// TwinCAT 3 PLC project _25_Memento
// ProgramVersion: 3.1.4023.0
// libraries:
//   Tc2_Standard, * (Beckhoff Automation GmbH)
//   Tc2_System, * (Beckhoff Automation GmbH)
//   Tc3_Module, * (Beckhoff Automation GmbH)
// project tree:
//   / MAIN.TcPOU, PlcTask.TcTTO
//   Memento Pattern/FBs/ RecipeEditor.TcPOU, Snapshot.TcPOU
//   Memento Pattern/ P_Memento.TcPOU
// (motion and I/O tree: see PLC project 13_decorator)
// real-time tasks:
//   TASK PlcTask: cycle T#10ms, priority 20, ADS port 350
// variable links:

CONFIGURATION _25_Memento
    RESOURCE PLC ON TwinCAT3
        TASK PlcTask(INTERVAL := T#10ms, PRIORITY := 20);
        PROGRAM P_Memento WITH PlcTask : P_Memento;
    END_RESOURCE
END_CONFIGURATION

// ---- Memento Pattern/P_Memento.TcPOU
PROGRAM P_Memento
VAR
	// Recipe editor and backup object
	pBackup : POINTER TO Snapshot;
	editor : RecipeEditor;
	
	// Recipe settings
	sTitle: STRING := 'Recipe 1';
	sRecipeSteps : ARRAY[1..5] OF STRING := ['Move Home', 'Move To Station A', 'Heater On', 'Apply Heat', 'Heater Off'];
	
	// Demo program control values
	bSetValues	: BOOL;
	bMakeBackup : BOOL;
	bRestore	: BOOL;
END_VAR

// Set the recipe values
IF bSetValues THEN
	bSetValues := FALSE;
	editor.setRecipe(sRecipeSteps);
	editor.setTitle(sTitle);
END_IF

// Make a backup at any time
IF bMakeBackup THEN
	bMakeBackup := FALSE;
	pBackup := editor.createSnapshot();
END_IF

// Restore to the backup state
IF bRestore AND (pBackup <> 0)THEN
	bRestore := FALSE;
	pBackup^.restore();
END_IF

END_PROGRAM

// ---- Memento Pattern/FBs/Snapshot.TcPOU
{attribute 'enable_dynamic_creation'}
FUNCTION_BLOCK Snapshot
VAR
	pEditor : POINTER TO RecipeEditor;
	sTitle : STRING;
	sRecipeSteps : ARRAY[1..5] OF STRING;
END_VAR

METHOD FB_exit : BOOL
VAR_INPUT
	bInCopyCode : BOOL; // if TRUE, the exit method is called for exiting an instance that is copied afterwards (online change).
END_VAR
// Clear the pointer on exit
IF pEditor <> 16#0000 THEN
	pEditor := 16#0000;
END_IF
END_METHOD

METHOD FB_init : BOOL
VAR_INPUT
	bInitRetains : BOOL; // if TRUE, the retain variables are initialized (warm start / cold start)
	bInCopyCode : BOOL;  // if TRUE, the instance afterwards gets moved into the copy code (online change)
	pEditor : POINTER TO RecipeEditor;
	sTitle : STRING;
	sRecipeSteps : ARRAY[1..5] OF STRING;
END_VAR
THIS^.pEditor := pEditor;
THIS^.sTitle := sTitle;
THIS^.sRecipeSteps := sRecipeSteps;
END_METHOD

METHOD restore
VAR_INPUT
END_VAR
pEditor^.setTitle(THIS^.sTitle);
pEditor^.setRecipe(THIS^.sRecipeSteps);
ADSLOGSTR( msgCtrlMask := ADSLOG_MSGTYPE_LOG, msgFmtStr := 'PLC Msg.: %s', strArg := 'Snapshot restored...');
END_METHOD

END_FUNCTION_BLOCK

// ---- Memento Pattern/FBs/RecipeEditor.TcPOU
FUNCTION_BLOCK RecipeEditor
VAR
	sTitle : STRING;
	sRecipeSteps : ARRAY[1..5] OF STRING;
	pSnapshot : POINTER TO Snapshot;
END_VAR

METHOD createSnapshot : POINTER TO Snapshot
VAR

END_VAR
IF THIS^.pSnapshot <> 0 THEN
	ADSLOGSTR( msgCtrlMask := ADSLOG_MSGTYPE_LOG, msgFmtStr := 'PLC Msg.: %s', strArg := 'Snapshot exists, deleting the old...');
	__DELETE(THIS^.pSnapshot);
END_IF


THIS^.pSnapshot := __NEW(Snapshot(pEditor := ADR(THIS^), sTitle := THIS^.sTitle, sRecipeSteps := THIS^.sRecipeSteps));
createSnapshot := THIS^.pSnapshot;
ADSLOGSTR( msgCtrlMask := ADSLOG_MSGTYPE_LOG, msgFmtStr := 'PLC Msg.: %s', strArg := 'New snapshot generated...');
END_METHOD

METHOD FB_exit : BOOL
VAR_INPUT
	bInCopyCode : BOOL; // if TRUE, the exit method is called for exiting an instance that is copied afterwards (online change).
END_VAR
// Clear the pointer on exit
IF THIS^.pSnapshot <> 0 THEN
	__DELETE(pSnapshot);
END_IF
END_METHOD

METHOD setRecipe
VAR_INPUT
	sRecipeSteps : ARRAY[1..5] OF STRING;
END_VAR
THIS^.sRecipeSteps := sRecipeSteps;
END_METHOD

METHOD setTitle
VAR_INPUT
	sTitle : STRING;
END_VAR
THIS^.sTitle := sTitle;
END_METHOD

END_FUNCTION_BLOCK

// ---- MAIN.TcPOU
PROGRAM MAIN
VAR
END_VAR

(* 
	GOF 		Without violating encapsulation, capture and externalize an object's internal state
				so that the object can be restored to this state later  
*)
P_Memento();

END_PROGRAM
